# EPICS alarm handler configuration: apps/alhConfig/beam_curr.alhConfig
GROUP    NULL                         BEAM_CURRENT
CHANNEL  BEAM_CURRENT                 hallb_IPM2C21A_CUR
$COMMAND  medm -x -attach -cmap -macro "sig=hallb_IPM2C21A_CUR" aiaocalc_alarm.adl >> /dev/null
$ALARMCOUNTFILTER  10 120
$GUIDANCE
              The beam current  measured at nA BPM 2C21A is out of spec.  Inform MCC about this.
$END
CHANNEL  BEAM_CURRENT                 hallb_IPM2C24A_CUR
$COMMAND  medm -x -attach -cmap -macro "sig=hallb_IPM2C24A_CUR" aiaocalc_alarm.adl >> /dev/null
$ALARMCOUNTFILTER  10 120
$GUIDANCE
              The beam current  measured at nA BPM 2C24A is out of spec.  Inform MCC about this.
$END
### CHANNEL  BEAM_CURRENT                 hallb_IPM2H01_CUR
### $COMMAND  medm -x -attach -cmap -macro "sig=hallb_IPM2H01_CUR" aiaocalc_alarm.adl >> /dev/null
### $ALARMCOUNTFILTER  10 120
### $GUIDANCE
###               The beam current  measured at nA BPM 2H01 is out of spec.  Inform MCC about this.
### $END
CHANNEL  BEAM_CURRENT                 scaler_calc1b
$COMMAND  medm -x -attach -cmap -macro "sig=scaler_calc1b" aiaocalc_alarm.adl >> /dev/null
$ALARMCOUNTFILTER  10 120
$GUIDANCE
              The beam current  measured by the Faraday Cup is out of spec.  Inform MCC about this.
$END

CHANNEL  BEAM_CURRENT                 scaler_eS5b
$COMMAND  medm -x -attach -cmap -macro "sig=scaler_eS5b" aiaocalc_alarm.adl >> /dev/null
$ALARMCOUNTFILTER  2 10
$GUIDANCE
              The downstream halo counter rate is above the spec. Beam needs some steering. Inform MCC about this.
$END

CHANNEL  BEAM_CURRENT   beam_stopper_alarm
$COMMAND  medm -x -attach -cmap -macro "sig=beam_stopper_alarm" aiaocalc_alarm.adl >> /dev/null
$ALARMCOUNTFILTER  -1 60
$GUIDANCE
              The beam stopper position and the beam current do not match. Beam stopper is supposed to be in the beam at high beam current reaching FCUP. Notify the BEAM EXPERT.
$END
